{attribute addProperty BoxType "EL3102-0000-0019"}
{attribute addProperty Id "AI_Standard_ChannelAT %I*ARRAY[0..2] OF AI_Standard_Channel_6D9FFE0F14818.50WcStateAT %I*WcState_98A4DF7520.250InfoDataAT %I*InfoData_BC63D37F80100"}
{attribute addProperty CRC "2850908330"}
{attribute addProperty SizeInBites "230"}
{attribute addProperty SizeInBytes "28.75"}
TYPE EL3102_8DA07E8B :
STRUCT
	{attribute addProperty Name "AI_Standard_Channel"}
	AI_Standard_Channel : ARRAY[0..2] OF AI_Standard_Channel_6D9FFE0F;
	{attribute addProperty Name "WcState"}
	WcState : WcState_98A4DF75;
	{attribute addProperty Name "InfoData"}
	InfoData : InfoData_BC63D37F;
END_STRUCT
END_TYPE

(* stored: Version 1.2.0.0, ProductVersion 3.1.4024.9
   DUT EL3102_8DA07E8B: Id {98badb98-2522-4a68-bf2e-94f0fa8a1cca} *)
